// Swaps values of to variables
FUNCTION Swap
VAR_IN_OUT
	Number1		: REAL;
	Number2		: REAL;
END_VAR
VAR
	Temp		: REAL;
END_VAR


// Just swap pointers
Temp := Number1;
Number1 := Number2;
Number2 := Temp;

END_FUNCTION

(* stored: Version 1.1.0.1, ProductVersion 3.1.4024.11
   POU Swap: Id {f2039616-09f6-4daf-a7c3-d64000caac91}, SpecialFunc None *)
